{attribute 'linkalways'} 
{attribute 'no_explicit_call' := 'This FB is a CLASS and must be accessed using methods or properties'}
{attribute 'enable_dynamic_creation'}
FUNCTION_BLOCK _ETcVnContourRetrievalMode EXTENDS EnumDatatypeBase
VAR
	localData : ETcVnContourRetrievalMode;
	activeData : REFERENCE TO ETcVnContourRetrievalMode;
	enumBaseDatatype : _DINT(localData);
END_VAR

METHOD PRIVATE AddLocalEnumeration
VAR_INPUT
	Enumeration : T_MAXSTRING;
	Value : ETcVnContourRetrievalMode;
END_VAR
AddEnumeration(Enumeration, Value);
END_METHOD

PROPERTY PUBLIC Address : PVOID
GET
Address := ADR(activeData);
END_GET
END_PROPERTY

METHOD PUBLIC ClearReference
VAR_INPUT
END_VAR
activeData REF= localData;
SetBaseDatatypeReference();
END_METHOD

METHOD PUBLIC Clone : I_Datatype
VAR
    pClone : POINTER TO _ETcVnContourRetrievalMode;
END_VAR
pClone := __NEW(_ETcVnContourRetrievalMode(InitialValue := Value));
Clone := pClone^;
END_METHOD

METHOD FB_init : BOOL
VAR_INPUT
	bInitRetains : BOOL; // if TRUE, the retain variables are initialized (warm start / cold start)
	bInCopyCode : BOOL;  // if TRUE, the instance afterwards gets moved into the copy code (online change)
	InitialValue : ETcVnContourRetrievalMode;
END_VAR
localData := InitialValue;
AddBaseDatatype(enumBaseDatatype);
ClearReference();

AddLocalEnumeration('TCVN_CRM_EXTERNAL', ETcVnContourRetrievalMode.TCVN_CRM_EXTERNAL);
AddLocalEnumeration('TCVN_CRM_LIST', ETcVnContourRetrievalMode.TCVN_CRM_LIST);
AddLocalEnumeration('TCVN_CRM_CONNECTED_COMPONENTS', ETcVnContourRetrievalMode.TCVN_CRM_CONNECTED_COMPONENTS);
AddLocalEnumeration('TCVN_CRM_TREE', ETcVnContourRetrievalMode.TCVN_CRM_TREE);
AddLocalEnumeration('TCVN_CRM_FLOODFILL', ETcVnContourRetrievalMode.TCVN_CRM_FLOODFILL);
END_METHOD

PROPERTY PUBLIC Identifier : T_MAXSTRING
GET
Identifier := 'ETcVnContourRetrievalMode';
END_GET
END_PROPERTY

METHOD IsEnumeratorValueEqual : BOOL
VAR_INPUT
	Enumerator : I_KeyValueForwardEnumerator;
END_VAR
VAR
	storedValue : ETcVnContourRetrievalMode;
END_VAR
IF NOT Enumerator.TryGet(storedValue) THEN
	RETURN;
END_IF

IsEnumeratorValueEqual := storedValue = activeData;
END_METHOD

METHOD PUBLIC MakeReferenceTo
VAR_INPUT
	ReferenceTarget : REFERENCE TO ETcVnContourRetrievalMode;
END_VAR
activeData REF= ReferenceTarget;
SetBaseDatatypeReference();
END_METHOD

METHOD PROTECTED SetBaseDatatypeReference
VAR_INPUT
END_VAR
enumBaseDatatype.MakeReferenceTo(activeData);
END_METHOD

PROPERTY PUBLIC Size : UDINT
GET
Size := SIZEOF(activeData);
END_GET
END_PROPERTY

METHOD TryMakeReferenceTo : BOOL
VAR_INPUT
	Target : I_Datatype;
END_VAR
VAR
	targetAsEnum : I_EnumDatatype;
	pTargetData : POINTER TO ETcVnContourRetrievalMode;
END_VAR
IF NOT Target.TryResolveAsEnumDatatype(targetAsEnum) THEN
	RETURN;
END_IF

IF targetAsEnum.Identifier <> Identifier THEN
	RETURN;
END_IF

pTargetData := Target.Address;
activeData REF= pTargetData^;
SetBaseDatatypeReference();
TryMakeReferenceTo := TRUE;
END_METHOD

PROPERTY PUBLIC Value : ETcVnContourRetrievalMode
GET
Value := activeData;
END_GET
SET
activeData := Value;
END_SET
END_PROPERTY

END_FUNCTION_BLOCK

(* stored: Version 1.1.0.1, ProductVersion 3.1.4024.12
   POU _ETcVnContourRetrievalMode: Id {3fa00f69-e8c8-42e5-8b19-c060885e3ea5}, SpecialFunc None
   Folder Constructor: Id {7cedbb3f-a3f7-4ff2-bb44-f594fb5a2cdd}
   Folder Private: Id {4250efb8-994f-412e-b156-9aefb89c62fc}
   Folder Protected: Id {0d771d95-df12-4ac2-aaab-97dca54d2441}
   Method AddLocalEnumeration: Id {b970629b-019d-4f76-bf9f-2215e5c8d914}
   Property Address: Id {31721e42-6b9f-4ca5-9f56-236511fac23d}
   Get Get: Id {dea5b6f4-8567-45e1-8014-79e480318664}
   Method ClearReference: Id {51d9ec53-786c-4600-8a1f-e4e0b569528b}
   Method Clone: Id {68f3cd62-127d-40f9-820e-d96e6d87550e}
   Method FB_init: Id {caa9dda7-1810-40c9-97e9-a69ded13314b}
   Property Identifier: Id {5cd1a69c-9ef6-4f52-8fda-bca15f9736ea}
   Get Get: Id {e0bbe87d-cbdb-41da-bbb1-45284a4e9db8}
   Method IsEnumeratorValueEqual: Id {7123e46b-59f1-4a4c-85f3-b9fa4968472a}
   Method MakeReferenceTo: Id {7cca9f60-cfcd-4e46-9f13-d2a9f94624aa}
   Method SetBaseDatatypeReference: Id {ef5da5e7-4701-4d8b-a6a1-98ba5a80ee65}
   Property Size: Id {8a3a7d46-c4a1-4a0d-969f-c5d3af061ca4}
   Get Get: Id {d07d3c03-df77-4316-ba2f-b8b97b6e6ea2}
   Method TryMakeReferenceTo: Id {0cc58875-ec17-41df-9c3a-930bdfe65bb3}
   Property Value: Id {8fa298df-af63-402e-a5b9-5a4a4e8e9456}
   Get Get: Id {0553fbf1-95fe-4bc7-8b71-ddf0f4a63cf3}
   Set Set: Id {98a31b8e-bb13-41cc-add6-56e5b6c13315} *)
